(* IEC 61131-3 sources: mocks/test/System/Timer, 3 files *)

(* ---- ConfigurableOffDelayMockTest.st ---- *)
USING System.Timer;
USING AxUnit.Assert;

NAMESPACE Simatic.Ax.Mocks
    /// Example function block that uses multiple OffDelay timers
    FUNCTION_BLOCK MultiOffDelayFunctionBlock
        VAR_INPUT
            enable1 : BOOL;
            enable2 : BOOL;
            enable3 : BOOL;
        END_VAR
        VAR_OUTPUT
            status1 : STRING;
            status2 : STRING;
            status3 : STRING;
        END_VAR
        VAR
            timer1 : OffDelay;
            timer2 : OffDelay;
            timer3 : OffDelay;
        END_VAR

        // Timer 1: 1 second delay
        timer1(signal := enable1, duration := T#1s);
        IF timer1.output THEN
            status1 := 'T1_ON';
        ELSE
            status1 := 'T1_OFF';
        END_IF;

        // Timer 2: 2 second delay
        timer2(signal := enable2, duration := T#2s);
        IF timer2.output THEN
            status2 := 'T2_ON';
        ELSE
            status2 := 'T2_OFF';
        END_IF;

        // Timer 3: 5 second delay
        timer3(signal := enable3, duration := T#5s);
        IF timer3.output THEN
            status3 := 'T3_ON';
        ELSE
            status3 := 'T3_OFF';
        END_IF;
    END_FUNCTION_BLOCK

    /// Test fixture demonstrating ConfigurableOffDelayMock usage
    {TestFixture}
    CLASS TestConfigurableOffDelayMock
        VAR
            testInstance, testInstanceStateless : MultiOffDelayFunctionBlock;
            payload, payloadStateless : ConfigurableOffDelayMockPayload;
        END_VAR

        /// Setup method to reset instances before each test
        {TestSetup}
        METHOD PUBLIC TestSetup
            payload := payloadStateless;
            testInstance := testInstanceStateless;
        END_METHOD

        /// Test with Timer 1 ON, Timer 2 OFF, Timer 3 ON
        /// Timers are identified by call order: 1st call = T1, 2nd call = T2, 3rd call = T3
        {Test}
        METHOD PUBLIC TestMultipleTimersWithDifferentStates
            // Reset counter before test
            payload.ResetCounter();

            // Configure payload: T1=TRUE, T2=FALSE, T3=TRUE (by call order)
            payload.T1_Enabled := TRUE;
            payload.T1_Output := TRUE;
            payload.T1_ElapsedTime := T#0ms;

            payload.T2_Enabled := TRUE;
            payload.T2_Output := FALSE;
            payload.T2_ElapsedTime := T#1s;

            payload.T3_Enabled := TRUE;
            payload.T3_Output := TRUE;
            payload.T3_ElapsedTime := T#0ms;

            // Apply mock with payload
            AxUnit.Mocking.Mock(
                mockeeFn := NAME_OF(OffDelay),
                mockFn := NAME_OF(ConfigurableOffDelayMock),
                payload := payload
            );

            // Execute function block
            // Timer calls happen in order: timer1 (1st call), timer2 (2nd call), timer3 (3rd call)
            testInstance(enable1 := FALSE, enable2 := FALSE, enable3 := FALSE);

            // Verify results
            Equal(expected := 'T1_ON', actual := testInstance.status1);
            Equal(expected := 'T2_OFF', actual := testInstance.status2);
            Equal(expected := 'T3_ON', actual := testInstance.status3);
        END_METHOD

        /// Test with all timers OFF (delay elapsed)
        {Test}
        METHOD PUBLIC TestAllTimersOff
            // Reset counter before test
            payload.ResetCounter();

            // Configure payload: All timers OFF
            payload.T1_Enabled := TRUE;
            payload.T1_Output := FALSE;
            payload.T1_ElapsedTime := T#1s;

            payload.T2_Enabled := TRUE;
            payload.T2_Output := FALSE;
            payload.T2_ElapsedTime := T#2s;

            payload.T3_Enabled := TRUE;
            payload.T3_Output := FALSE;
            payload.T3_ElapsedTime := T#5s;

            // Apply mock with payload
            AxUnit.Mocking.Mock(
                mockeeFn := NAME_OF(OffDelay),
                mockFn := NAME_OF(ConfigurableOffDelayMock),
                payload := payload
            );

            // Execute function block
            testInstance(enable1 := FALSE, enable2 := FALSE, enable3 := FALSE);

            // Verify results
            Equal(expected := 'T1_OFF', actual := testInstance.status1);
            Equal(expected := 'T2_OFF', actual := testInstance.status2);
            Equal(expected := 'T3_OFF', actual := testInstance.status3);
        END_METHOD

        /// Test with only Timer 2 enabled (2nd call)
        {Test}
        METHOD PUBLIC TestOnlyTimer2Enabled
            // Reset counter before test
            payload.ResetCounter();

            // Configure payload: Only T2 enabled and ON
            payload.T1_Enabled := FALSE;  // 1st call returns FALSE

            payload.T2_Enabled := TRUE;   // 2nd call returns TRUE
            payload.T2_Output := TRUE;
            payload.T2_ElapsedTime := T#0ms;

            payload.T3_Enabled := FALSE;  // 3rd call returns FALSE

            // Apply mock with payload
            AxUnit.Mocking.Mock(
                mockeeFn := NAME_OF(OffDelay),
                mockFn := NAME_OF(ConfigurableOffDelayMock),
                payload := payload
            );

            // Execute function block
            testInstance(enable1 := FALSE, enable2 := FALSE, enable3 := FALSE);

            // Verify results
            Equal(expected := 'T1_OFF', actual := testInstance.status1); // 1st call: not enabled
            Equal(expected := 'T2_ON', actual := testInstance.status2);  // 2nd call: enabled and TRUE
            Equal(expected := 'T3_OFF', actual := testInstance.status3); // 3rd call: not enabled
        END_METHOD

        /// Test with all timers ON (signal still active)
        {Test}
        METHOD PUBLIC TestAllTimersOn
            // Reset counter before test
            payload.ResetCounter();

            // Configure payload: All timers ON
            payload.T1_Enabled := TRUE;
            payload.T1_Output := TRUE;
            payload.T1_ElapsedTime := T#0ms;

            payload.T2_Enabled := TRUE;
            payload.T2_Output := TRUE;
            payload.T2_ElapsedTime := T#0ms;

            payload.T3_Enabled := TRUE;
            payload.T3_Output := TRUE;
            payload.T3_ElapsedTime := T#0ms;

            // Apply mock with payload
            AxUnit.Mocking.Mock(
                mockeeFn := NAME_OF(OffDelay),
                mockFn := NAME_OF(ConfigurableOffDelayMock),
                payload := payload
            );

            // Execute function block
            testInstance(enable1 := TRUE, enable2 := TRUE, enable3 := TRUE);

            // Verify results
            Equal(expected := 'T1_ON', actual := testInstance.status1);
            Equal(expected := 'T2_ON', actual := testInstance.status2);
            Equal(expected := 'T3_ON', actual := testInstance.status3);
        END_METHOD
    END_CLASS
END_NAMESPACE

(* ---- ConfigurableOnDelayMockTest.st ---- *)
USING System.Timer;
USING AxUnit.Assert;

NAMESPACE Simatic.Ax.Mocks
    /// Example function block that uses multiple OnDelay timers
    FUNCTION_BLOCK MultiTimerFunctionBlock
        VAR_INPUT
            enable1 : BOOL;
            enable2 : BOOL;
            enable3 : BOOL;
        END_VAR
        VAR_OUTPUT
            status1 : STRING;
            status2 : STRING;
            status3 : STRING;
        END_VAR
        VAR
            timer1 : OnDelay;
            timer2 : OnDelay;
            timer3 : OnDelay;
        END_VAR

        // Timer 1: 1 second delay
        timer1(signal := enable1, duration := T#1s);
        IF timer1.output THEN
            status1 := 'T1_ELAPSED';
        ELSE
            status1 := 'T1_WAITING';
        END_IF;

        // Timer 2: 2 second delay
        timer2(signal := enable2, duration := T#2s);
        IF timer2.output THEN
            status2 := 'T2_ELAPSED';
        ELSE
            status2 := 'T2_WAITING';
        END_IF;

        // Timer 3: 5 second delay
        timer3(signal := enable3, duration := T#5s);
        IF timer3.output THEN
            status3 := 'T3_ELAPSED';
        ELSE
            status3 := 'T3_WAITING';
        END_IF;
    END_FUNCTION_BLOCK

    /// Test fixture demonstrating ConfigurableOnDelayMock usage
    {TestFixture}
    CLASS TestConfigurableOnDelayMock
        VAR
            testInstance, testInstanceStateless : MultiTimerFunctionBlock;
            payload, payloadStateless : ConfigurableOnDelayMockPayload;
        END_VAR

        /// Setup method to reset instances before each test
        {TestSetup}
        METHOD PUBLIC TestSetup
            payload := payloadStateless;
            testInstance := testInstanceStateless;
        END_METHOD

        /// Test with Timer 1 elapsed, Timer 2 waiting, Timer 3 elapsed
        /// Timers are identified by call order: 1st call = T1, 2nd call = T2, 3rd call = T3
        {Test}
        METHOD PUBLIC TestMultipleTimersWithDifferentStates
            // Reset counter before test
            payload.ResetCounter();

            // Configure payload: T1=TRUE, T2=FALSE, T3=TRUE (by call order)
            payload.T1_Enabled := TRUE;
            payload.T1_Output := TRUE;
            payload.T1_ElapsedTime := T#1s;

            payload.T2_Enabled := TRUE;
            payload.T2_Output := FALSE;
            payload.T2_ElapsedTime := T#500ms;

            payload.T3_Enabled := TRUE;
            payload.T3_Output := TRUE;
            payload.T3_ElapsedTime := T#5s;

            // Apply mock with payload
            AxUnit.Mocking.Mock(
                mockeeFn := NAME_OF(OnDelay),
                mockFn := NAME_OF(ConfigurableOnDelayMock),
                payload := payload
            );

            // Execute function block
            // Timer calls happen in order: timer1 (1st call), timer2 (2nd call), timer3 (3rd call)
            testInstance(enable1 := TRUE, enable2 := TRUE, enable3 := TRUE);

            // Verify results
            Equal(expected := 'T1_ELAPSED', actual := testInstance.status1);
            Equal(expected := 'T2_WAITING', actual := testInstance.status2);
            Equal(expected := 'T3_ELAPSED', actual := testInstance.status3);
        END_METHOD

        /// Test with all timers elapsed
        {Test}
        METHOD PUBLIC TestAllTimersElapsed
            // Reset counter before test
            payload.ResetCounter();

            // Configure payload: All timers elapsed
            payload.T1_Enabled := TRUE;
            payload.T1_Output := TRUE;
            payload.T1_ElapsedTime := T#1s;

            payload.T2_Enabled := TRUE;
            payload.T2_Output := TRUE;
            payload.T2_ElapsedTime := T#2s;

            payload.T3_Enabled := TRUE;
            payload.T3_Output := TRUE;
            payload.T3_ElapsedTime := T#5s;

            // Apply mock with payload
            AxUnit.Mocking.Mock(
                mockeeFn := NAME_OF(OnDelay),
                mockFn := NAME_OF(ConfigurableOnDelayMock),
                payload := payload
            );

            // Execute function block
            testInstance(enable1 := TRUE, enable2 := TRUE, enable3 := TRUE);

            // Verify results
            Equal(expected := 'T1_ELAPSED', actual := testInstance.status1);
            Equal(expected := 'T2_ELAPSED', actual := testInstance.status2);
            Equal(expected := 'T3_ELAPSED', actual := testInstance.status3);
        END_METHOD

        /// Test with only Timer 2 enabled (2nd call)
        {Test}
        METHOD PUBLIC TestOnlyTimer2Enabled
            // Reset counter before test
            payload.ResetCounter();

            // Configure payload: Only T2 enabled and elapsed
            payload.T1_Enabled := FALSE;  // 1st call returns FALSE

            payload.T2_Enabled := TRUE;   // 2nd call returns TRUE
            payload.T2_Output := TRUE;
            payload.T2_ElapsedTime := T#2s;

            payload.T3_Enabled := FALSE;  // 3rd call returns FALSE

            // Apply mock with payload
            AxUnit.Mocking.Mock(
                mockeeFn := NAME_OF(OnDelay),
                mockFn := NAME_OF(ConfigurableOnDelayMock),
                payload := payload
            );

            // Execute function block
            testInstance(enable1 := TRUE, enable2 := TRUE, enable3 := TRUE);

            // Verify results
            Equal(expected := 'T1_WAITING', actual := testInstance.status1); // 1st call: not enabled
            Equal(expected := 'T2_ELAPSED', actual := testInstance.status2); // 2nd call: enabled and TRUE
            Equal(expected := 'T3_WAITING', actual := testInstance.status3); // 3rd call: not enabled
        END_METHOD
    END_CLASS
END_NAMESPACE

(* ---- IdentifierBasedOnDelayMockTest.st ---- *)
USING System.Timer;
USING AxUnit.Assert;

NAMESPACE Simatic.Ax.Mocks
    /// Example function block with conditional timer usage
    /// Depending on mode, different timers are called at different positions
    FUNCTION_BLOCK ConditionalTimerExample
        VAR_INPUT
            mode : INT;         // 1 = use T1+T2, 2 = use T1+T3
            enable : BOOL;
        END_VAR
        VAR_OUTPUT
            status : STRING;
        END_VAR
        VAR
            timer1 : OnDelay;   // Always used at position 1
            timer2 : OnDelay;   // Used at position 2 in mode 1
            timer3 : OnDelay;   // Used at position 2 in mode 2
        END_VAR

        // Timer 1 is always called first (position 1)
        timer1(signal := enable, duration := T#1s);

        IF mode = 1 THEN
            // Mode 1: Timer 2 is called at position 2
            timer2(signal := enable, duration := T#2s);

            IF timer1.output AND timer2.output THEN
                status := 'MODE1_BOTH_ELAPSED';
            ELSIF timer1.output THEN
                status := 'MODE1_T1_ELAPSED';
            ELSE
                status := 'MODE1_WAITING';
            END_IF;

        ELSIF mode = 2 THEN
            // Mode 2: Timer 3 is called at position 2
            timer3(signal := enable, duration := T#3s);

            IF timer1.output AND timer3.output THEN
                status := 'MODE2_BOTH_ELAPSED';
            ELSIF timer1.output THEN
                status := 'MODE2_T1_ELAPSED';
            ELSE
                status := 'MODE2_WAITING';
            END_IF;
        END_IF;
    END_FUNCTION_BLOCK

    /// Test fixture demonstrating IdentifierBasedTimerMock with conditional timers
    {TestFixture}
    CLASS TestIdentifierBasedOnDelayMock
        VAR
            testInstance, testInstanceStateless : ConditionalTimerExample;
            testInstanceMulti, testInstanceMultiStateless : MultiTimerFunctionBlock;
            payload, payloadStateless : IdentifierBasedOnDelayMockPayload;
        END_VAR

        {TestSetup}
        METHOD PUBLIC TestSetup
            payload := payloadStateless;
            testInstance := testInstanceStateless;
            testInstanceMulti := testInstanceMultiStateless;
        END_METHOD

        /// Test Mode 1: T1 at position 1, T2 at position 2
        {Test}
        METHOD PUBLIC TestMode1_BothTimersElapsed
            payload.ResetCounter();

            // Timer 1: Position 1 (always first call)
            payload.T1_Enabled := TRUE;
            payload.T1_CallPosition := 1;  // 1st call
            payload.T1_Output := TRUE;
            payload.T1_ElapsedTime := T#1s;

            // Timer 2: Position 2 (second call in mode 1)
            payload.T2_Enabled := TRUE;
            payload.T2_CallPosition := 2;  // 2nd call
            payload.T2_Output := TRUE;
            payload.T2_ElapsedTime := T#2s;

            // Timer 3: not called in mode 1
            payload.T3_Enabled := FALSE;

            // Apply mock
            AxUnit.Mocking.Mock(
                mockeeFn := NAME_OF(OnDelay),
                mockFn := NAME_OF(IdentifierBasedOnDelayMock),
                payload := payload
            );

            // Execute in mode 1
            testInstance(mode := 1, enable := TRUE);

            // Verify both timers elapsed
            Equal(expected := 'MODE1_BOTH_ELAPSED', actual := testInstance.status);
        END_METHOD

        /// Test Mode 1: T1 elapsed, T2 waiting
        {Test}
        METHOD PUBLIC TestMode1_OnlyT1Elapsed
            payload.ResetCounter();

            // Timer 1: Position 1, elapsed
            payload.T1_Enabled := TRUE;
            payload.T1_CallPosition := 1;
            payload.T1_Output := TRUE;
            payload.T1_ElapsedTime := T#1s;

            // Timer 2: Position 2, not elapsed
            payload.T2_Enabled := TRUE;
            payload.T2_CallPosition := 2;
            payload.T2_Output := FALSE;
            payload.T2_ElapsedTime := T#500ms;

            // Timer 3: not called in mode 1
            payload.T3_Enabled := FALSE;

            // Apply mock
            AxUnit.Mocking.Mock(
                mockeeFn := NAME_OF(OnDelay),
                mockFn := NAME_OF(IdentifierBasedOnDelayMock),
                payload := payload
            );

            // Execute in mode 1
            testInstance(mode := 1, enable := TRUE);

            // Verify only T1 elapsed
            Equal(expected := 'MODE1_T1_ELAPSED', actual := testInstance.status);
        END_METHOD

        /// Test Mode 2: T1 at position 1, T3 at position 2
        {Test}
        METHOD PUBLIC TestMode2_BothTimersElapsed
            payload.ResetCounter();

            // Timer 1: Position 1 (always first call)
            payload.T1_Enabled := TRUE;
            payload.T1_CallPosition := 1;  // 1st call
            payload.T1_Output := TRUE;
            payload.T1_ElapsedTime := T#1s;

            // Timer 2: not called in mode 2
            payload.T2_Enabled := FALSE;

            // Timer 3: Position 2 (second call in mode 2)
            payload.T3_Enabled := TRUE;
            payload.T3_CallPosition := 2;  // 2nd call
            payload.T3_Output := TRUE;
            payload.T3_ElapsedTime := T#3s;

            // Apply mock
            AxUnit.Mocking.Mock(
                mockeeFn := NAME_OF(OnDelay),
                mockFn := NAME_OF(IdentifierBasedOnDelayMock),
                payload := payload
            );

            // Execute in mode 2
            testInstance(mode := 2, enable := TRUE);

            // Verify both timers elapsed
            Equal(expected := 'MODE2_BOTH_ELAPSED', actual := testInstance.status);
        END_METHOD

        /// Test Mode 2: T1 elapsed, T3 waiting
        {Test}
        METHOD PUBLIC TestMode2_OnlyT1Elapsed
            payload.ResetCounter();

            // Timer 1: Position 1, elapsed
            payload.T1_Enabled := TRUE;
            payload.T1_CallPosition := 1;
            payload.T1_Output := TRUE;
            payload.T1_ElapsedTime := T#1s;

            // Timer 2: not called in mode 2
            payload.T2_Enabled := FALSE;

            // Timer 3: Position 2, not elapsed
            payload.T3_Enabled := TRUE;
            payload.T3_CallPosition := 2;
            payload.T3_Output := FALSE;
            payload.T3_ElapsedTime := T#1500ms;

            // Apply mock
            AxUnit.Mocking.Mock(
                mockeeFn := NAME_OF(OnDelay),
                mockFn := NAME_OF(IdentifierBasedOnDelayMock),
                payload := payload
            );

            // Execute in mode 2
            testInstance(mode := 2, enable := TRUE);

            // Verify only T1 elapsed
            Equal(expected := 'MODE2_T1_ELAPSED', actual := testInstance.status);
        END_METHOD

        /// Test with 3 sequential timers (no conditional logic)
        {Test}
        METHOD PUBLIC TestSequentialTimers
            payload.ResetCounter();

            // Configure 3 timers at positions 1, 2, 3
            payload.T1_Enabled := TRUE;
            payload.T1_CallPosition := 1;
            payload.T1_Output := TRUE;
            payload.T1_ElapsedTime := T#1s;

            payload.T2_Enabled := TRUE;
            payload.T2_CallPosition := 2;
            payload.T2_Output := FALSE;
            payload.T2_ElapsedTime := T#500ms;

            payload.T3_Enabled := TRUE;
            payload.T3_CallPosition := 3;
            payload.T3_Output := TRUE;
            payload.T3_ElapsedTime := T#5s;

            // Apply mock
            AxUnit.Mocking.Mock(
                mockeeFn := NAME_OF(OnDelay),
                mockFn := NAME_OF(IdentifierBasedOnDelayMock),
                payload := payload
            );

            // Execute
            testInstanceMulti(enable1 := TRUE, enable2 := TRUE, enable3 := TRUE);

            // Verify results
            Equal(expected := 'T1_ELAPSED', actual := testInstanceMulti.status1);
            Equal(expected := 'T2_WAITING', actual := testInstanceMulti.status2);
            Equal(expected := 'T3_ELAPSED', actual := testInstanceMulti.status3);
        END_METHOD
    END_CLASS
END_NAMESPACE
